TYPE DUT_HMI_08_MANUALS :
STRUCT
	PS : ARRAY[0..CNC.NUM_MAX_MANUALS_08-1] OF BOOL;
	LS : ARRAY[0..CNC.NUM_MAX_MANUALS_08-1] OF BOOL;
END_STRUCT
END_TYPE

(* stored: Version 1.1.0.1, ProductVersion 3.1.4024.13
   DUT DUT_HMI_08_MANUALS: Id {9efdb397-5732-4e87-aaf5-dcf020809a9d} *)
